(* CoDeSys 2.3.9.48 project: test_CHP_switch.pro *)
(* Libraries: Standard.lib 20.5.14 07:13:26, Iecsfc.lib 30.1.13 12:05:12, SYSLIBCALLBACK.LIB 30.1.13 12:05:12 *)

(* PLC configuration (modules and I/O channels)
K-Bus [K_Bus] node 0, in %IB0 out %QB0 {KbusBusMode = 1; KbusCycleTime = 10000; KbusThreadPriority = 0; KbusSetOutputsToZeroOnApplicationStop = 1}
IEC60870-5-Konfig [IEC60870_Konfig] node 1, in %IB10000 out %QB10000 {IEC870_tAFZ_Kurz = t#500ms; IEC870_tAFZ_Lang = t#5s; IEC870_tAFZ_Default = t#2s; IEC870_nMaxTLGBufferSize = 32; IEC870_xUseSNTP = 1; IEC870_byTaskPrio = 7; IEC870_tTaskTime = t#20ms; IEC870_byTaskPrio = 8; IEC870_tTaskTime = t#20ms; IEC870_byTaskPrio = 9; IEC870_tTaskTime = t#20ms; IEC870_byTaskPrio = 10; IEC870_tTaskTime = t#20ms; IEC870_byVarGenMode = 1; IEC870_sSelSprache = DEUTSCH; IEC870_sTargetTyp = 758-8xx; IEC870_sUsedLib = Standard.LIB; IEC870_sUsedLib = SysLibCallback.LIB; IEC870_sUsedLib = SysLibRtc.LIB; IEC870_sUsedLib = SysLibSockets.LIB; IEC870_sUsedLib = SysLibMem.LIB; IEC870_sUsedLib = SysLibTime.LIB; IEC870_sUsedLib = SysLibSem.LIB; IEC870_sUsedLib = SysLibCom.LIB; IEC870_sInputAdr640 = %IB0; IEC870_sOutputAdr640 = %QB0; IEC870_UsedInfoObjFB_V2 = TRUE; IEC870_NTP_ServerAdress = 192.53.103.108; IEC870_NTP_RequestResponseTime = t#50ms; IEC870_NTP_UpdateIntervall = 60; IEC870_NTP_WatchdogTime = 10; IEC870_sUsedLib = SerComm.LIB; IEC870_sUsedLib = WagoLibEthernet_01.lib; IEC870_sUsedLib = WagoLibSntp.LIB; IEC870_sUsedLib = WagoLibNTP.LIB; IEC870_sUsedLib = WagoLibPing.lib; IEC870_sUsedLib = WagoLib60870Base.lib; IEC870_sUsedLib = WagoLib60870Slave.lib; IEC870_sUsedLib = WagoLib60870Master.lib; gsiIEC870_CLOCK_TimeZone = 0; gnIEC870_CLOCK_DST_Mode = 0; IEC870_xZW_SendSpoantan = 0; IEC870_diTimeOutC_Objs = 1000; IEC870_diHistBufferSize = 16; IEC870_xEnableGaForCpObj = 1; IEC870_byParameter = 0; IEC870_diParameter = 0; IEC870_diParameter = 0; IEC870_diParameter = 0; IEC870_byParameter = 0; IEC870_byParameter = 0; IEC870_byParameter = 0; IEC870_sParameter = 0; IEC870_sParameter = 0; IEC870_sParameter = 0}
Modbus variables [PFC200MODBUS] node 2, in %IB0 out %QB0 {PlcStopBehaviour = 1; FiledbusErrorBehaviour = 1; TcpOperation = 1; TcpPort = 502; TcpTimeout = 600; UdpOperation = 1; UdpPort = 502; RtuOperation = 0; NodeId = 1; ResponseTimeout = 5000; Interface = 0; Baud = 115200; StopBits = 1; Parity = 1; FlowCtrl = 0; PhysInterface = 0}
IEC61850-Konfig [IEC61850_Konfig] node 3, in %IB10000 out %QB10000 {IEC61850_sSelSprache = DEUTSCH; IEC61850_sTargetTyp = 758-8xx}
DNP3-Konfig [DNP3_Konfig] node 4, in %IB10000 out %QB10000 {IEC61850_sSelSprache = DEUTSCH; IEC61850_sTargetTyp = 758-8xx}
Modbus-Master [MB_MASTER] node 5, in %IB0 out %QB0
*)

(* Task configuration *)
TASK NewTask (PRIORITY := 31, INTERVAL := T#1000ms);
	PLC_PRG(b_fb_gridbus_request:= , b_fb_batbus_request:= , b_batbus_close_request=> , b_gridbus_close_request=> );
END_TASK

(* Global variable list: Global_Variables *)
VAR_GLOBAL

(* TEST SETTINGS CHP SWICHT HANDLER *)

	Grid_IN: BOOL;
	BAT_out: BOOL;
	Grid_OUT: BOOL;
	BAT_IN: BOOL;

	Group1_3F_Selector_auto_bus_select:BOOL;
	CHP_control_internal_contacter_switch_state: BOOL;
	Group1_3F_relay_state_battery_bus : BOOL;
	Group1_3F_relay_state_grid_bus :BOOL;
	CHP_control_Offgrid_request : BOOL;
END_VAR

(* POU 04. Frequency based Bus Select/PLC_PRG, ST *)
PROGRAM PLC_PRG
VAR_INPUT

	b_fb_gridbus_request							:	BOOL; (* request based on frequency, has delayed switching!! *)
	b_fb_batbus_request								:	BOOL; (* request based on frequency, has delayed switching!! *)

END_VAR

VAR_OUTPUT

	b_batbus_close_request							:	BOOL; (* request based on frequency, has delayed switching!! *)
	b_gridbus_close_request							:	BOOL; (* request based on frequency, has delayed switching!! *)

END_VAR
VAR
	z: INT;
	y: BOOL;
END_VAR
(* CHP handler uses frequency based switching input to control real CHP swithcing when auto input is high *)
(* CHP handler delays switching, such that the CHP can depower and disconnect before switch *)
(* CHP handler delays on-switching, making sure the CHP is disconnected. *)
(* CHP handler delays on-switching, making sure the CHP will connect to the right bus (in the right mode). *)

(* ____________________________  AUTO SWITCH CONTROL  ___________________________ *)
IF (Group1_3F_Selector_auto_bus_select = TRUE) THEN

	(*check if wanted state to CHP signal is right, change when required *)
	IF (b_fb_gridbus_request =TRUE AND b_fb_batbus_request =FALSE)  THEN
		CHP_control_Offgrid_request :=FALSE;
		z :=0;
		y := FALSE;
	ELSIF (b_fb_batbus_request =TRUE)  THEN
		CHP_control_Offgrid_request :=TRUE;
		z := 100;
		y := TRUE;
	ELSE
		z := 50;
	END_IF;
(*
IF (b_fb_batbus_request )  THEN
		CHP_control_Offgrid_request :=TRUE;
		z :=0;
		y := FALSE;
	ELSE
		z :=50;
		IF (b_fb_gridbus_request =TRUE)  THEN
		CHP_control_Offgrid_request :=FALSE;
		z := 100;
		y := TRUE;
		END_IF;
	END_IF;*)
z := z + 1;

	(* perform switch between busses when CHP has disconnceted *)
	IF (CHP_control_internal_contacter_switch_state =FALSE) THEN

		(* Close bat relais when grid relais is open en bat request is still true*)
		IF (b_fb_batbus_request =TRUE) THEN
			b_gridbus_close_request := FALSE; (* Disconnect GRID SCWICH*)
			IF (Group1_3F_relay_state_grid_bus = FALSE) THEN
				b_batbus_close_request := TRUE;
			END_IF;
		END_IF;

		(* Close grid relais when bat relais is open en grid request is still true*)
		IF (b_fb_gridbus_request =TRUE) THEN
			b_batbus_close_request := FALSE; (* Disconnect *)
			IF (Group1_3F_relay_state_battery_bus =FALSE) THEN
				b_gridbus_close_request := TRUE;
			END_IF;
		END_IF;
	END_IF;


(* ____________________________  MANUAL CONTROL  ___________________________ *)
ELSE
	z := 200;
	(* check if batbus relais is closed, if so, request offgrid (via wanted state *)
	IF (Group1_3F_relay_state_battery_bus =TRUE) THEN
		CHP_control_Offgrid_request :=TRUE;
	ELSE (* IF Group1_3F_relay_state_grid_bus THEN *)
		CHP_control_Offgrid_request :=FALSE;
	END_IF;
END_IF;
END_PROGRAM

(* POU 04. Frequency based Bus Select/test_switch, LD *)
PROGRAM test_switch
VAR
	test: CHP_Switch_Handler;
END_VAR
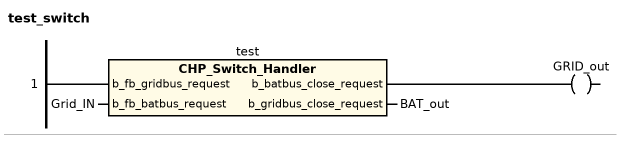
_LD_ (* Ladder Diagram *)
NETWORK 1
	test:CHP_Switch_Handler(b_fb_gridbus_request: *, b_fb_batbus_request: Grid_IN, b_gridbus_close_request => BAT_out) --- (GRID_out)
_END_LD_
(* the same logic as Structured Text *)
(* Network 1 *)
test(b_fb_gridbus_request := TRUE, b_fb_batbus_request := Grid_IN);
BAT_out := test.b_gridbus_close_request;
GRID_out := test.b_batbus_close_request;
END_PROGRAM

(* POU 04. Frequency based Bus Select/CHP_Switch_Handler, ST *)
FUNCTION_BLOCK CHP_Switch_Handler

VAR_INPUT

	b_fb_gridbus_request							:	BOOL; (* request based on frequency, has delayed switching!! *)
	b_fb_batbus_request								:	BOOL; (* request based on frequency, has delayed switching!! *)

END_VAR

VAR_OUTPUT

	b_batbus_close_request							:	BOOL; (* request based on frequency, has delayed switching!! *)
	b_gridbus_close_request							:	BOOL; (* request based on frequency, has delayed switching!! *)

END_VAR

VAR
(* ____________________________  USED GLOBAL VARIABLES  ___________________________ *)
(*
	(* INPUTS *)
	CHP_control_internal_contacter_switch_state  			AT %IX121.15 : BOOL;
	Group1_3F_Selector_auto_bus_select    				AT %IX121.2 : BOOL;
	Group1_3F_relay_state_battery_bus   					AT %IX120.1  : BOOL;
	Group1_3F_relay_state_grid_bus   						AT %IX120.0  : BOOL;

	(* OUTPUTS *)
	Group1_3F_Auto_relay_control_battery_bus   			AT %QX128.1  : BOOL;
	Group1_3F_Auto_relay_control_grid_bus   				AT %QX128.0  : BOOL;
	CHP_control_Offgrid_request    							AT %QX129.4  : BOOL;
*)
	y: BOOL := FALSE;
	z: INT :=0;
END_VAR
(* CHP handler uses frequency based switching input to control real CHP swithcing when auto input is high *)
(* CHP handler delays switching, such that the CHP can depower and disconnect before switch *)
(* CHP handler delays on-switching, making sure the CHP is disconnected. *)
(* CHP handler delays on-switching, making sure the CHP will connect to the right bus (in the right mode). *)

(* ____________________________  AUTO SWITCH CONTROL  ___________________________ *)
IF (Group1_3F_Selector_auto_bus_select = TRUE) THEN

	(*check if wanted state to CHP signal is right, change when required *)
	IF (b_fb_gridbus_request =TRUE AND b_fb_batbus_request =FALSE)  THEN
		CHP_control_Offgrid_request :=FALSE;
		z :=0;
		y := FALSE;
	ELSIF (b_fb_batbus_request =TRUE)  THEN
		CHP_control_Offgrid_request :=TRUE;
		z := 100;
		y := TRUE;
	ELSE
		z := 50;
	END_IF;
(*
IF (b_fb_batbus_request )  THEN
		CHP_control_Offgrid_request :=TRUE;
		z :=0;
		y := FALSE;
	ELSE
		z :=50;
		IF (b_fb_gridbus_request =TRUE)  THEN
		CHP_control_Offgrid_request :=FALSE;
		z := 100;
		y := TRUE;
		END_IF;
	END_IF;*)
z := z + 1;

	(* perform switch between busses when CHP has disconnceted *)
(*	IF (CHP_control_internal_contacter_switch_state =FALSE) THEN

		(* Close bat relais when grid relais is open en bat request is still true*)
		IF (b_fb_batbus_request =TRUE) THEN
			b_gridbus_close_request := FALSE; (* Disconnect GRID SCWICH*)
			IF (Group1_3F_relay_state_grid_bus = FALSE) THEN
				b_batbus_close_request := TRUE;
			END_IF;
		END_IF;

		(* Close grid relais when bat relais is open en grid request is still true*)
		IF (b_fb_gridbus_request =TRUE) THEN
			b_batbus_close_request := FALSE; (* Disconnect *)
			IF (Group1_3F_relay_state_battery_bus =FALSE) THEN
				b_gridbus_close_request := TRUE;
			END_IF;
		END_IF;
	END_IF;

*)
(* ____________________________  MANUAL CONTROL  ___________________________ *)
ELSE
	z := 200;
	(* check if batbus relais is closed, if so, request offgrid (via wanted state *)
	IF (Group1_3F_relay_state_battery_bus =TRUE) THEN
		CHP_control_Offgrid_request :=TRUE;
	ELSE (* IF Group1_3F_relay_state_grid_bus THEN *)
		CHP_control_Offgrid_request :=FALSE;
	END_IF;
END_IF;
END_FUNCTION_BLOCK
